SUBAPPLICATION Uebung_004d_T (* Exercise for FB_T_FF (Toggle Flip-Flop) *)
  (* Standard: 61499-2; Description: Copyright (c) 2026 Meisterschulen am Ostbahnhof *)
  (* Version 1.0, 2026-05-07, Gemini CLI, Meisterschulen am Ostbahnhof *)
  PACKAGE Uebungen;
  IMPORT logiBUS::io::DI::logiBUS_DI::Input_I1;
  IMPORT logiBUS::io::DI::logiBUS_DI::Input_I2;
  IMPORT logiBUS::io::DQ::logiBUS_DO::Output_Q1;
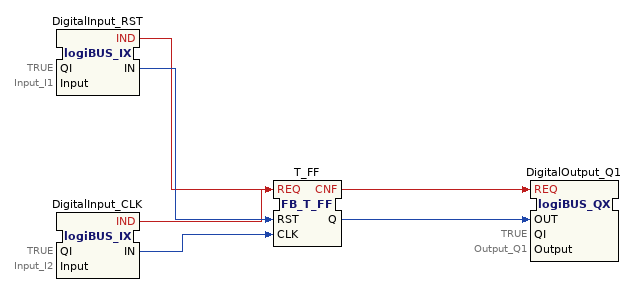
  FBS
    DigitalInput_RST : logiBUS::io::DI::logiBUS_IX(QI := TRUE, Input := Input_I1);
    DigitalInput_CLK : logiBUS::io::DI::logiBUS_IX(QI := TRUE, Input := Input_I2);
    T_FF : logiBUS::bistableElements::FB_T_FF;
    DigitalOutput_Q1 : logiBUS::io::DQ::logiBUS_QX(QI := TRUE, Output := Output_Q1);
  END_FBS
  EVENT_CONNECTIONS
    DigitalInput_RST.IND TO T_FF.REQ;
    DigitalInput_CLK.IND TO T_FF.REQ;
    T_FF.CNF TO DigitalOutput_Q1.REQ;
  END_CONNECTIONS
  DATA_CONNECTIONS
    DigitalInput_RST.IN TO T_FF.RST;
    DigitalInput_CLK.IN TO T_FF.CLK;
    T_FF.Q TO DigitalOutput_Q1.OUT;
  END_CONNECTIONS
END_SUBAPPLICATION
